{attribute 'OPC.UA.DA.StructuredType' := '1'}
TYPE SRecoveryRequestOutput EXTENDS STriggeredOutput :
STRUCT
	RequestedState: STRING(256);
END_STRUCT
END_TYPE

(* stored: Version 1.1.0.1
   DUT SRecoveryRequestOutput: Id {282aac72-0a3e-4332-9c40-eec7c0fb124d} *)
